{attribute addProperty BoxType "EK1100-0000-0018"}
{attribute addProperty Id "Beckhoff_ER3xxxEK1122Beckhoff_ER3xxxEK1122_CD7314C73040380"}
{attribute addProperty CRC "4196660496"}
{attribute addProperty SizeInBites "3040"}
{attribute addProperty SizeInBytes "380"}
TYPE Beckhoff_ER3xxx_FA23F510 EXTENDS EK1100_179A0949 :
STRUCT
	{attribute addProperty Name "Beckhoff_ER3xxxEK1122"}
	Beckhoff_ER3xxxEK1122 : Beckhoff_ER3xxxEK1122_CD7314C7;
END_STRUCT
END_TYPE

(* stored: Version 1.2.0.0, ProductVersion 3.1.4024.9
   DUT Beckhoff_ER3xxx_FA23F510: Id {22a4da82-bd3c-4399-966d-1a745c0179ec} *)
